Fanuc KAREL source: kc00004.KL

-- PROVISIONAL review KL for V1013-1; original PC SHA256 3c03b46ae540357a8fdae369b7eedd962a0a2d7ad2d21525eb34883495ea0831
-- Incomplete behavior may be omitted. Consult companion uncertainty JSON. Do not deploy.
PROGRAM KC00004
%NOLOCKGROUP
BEGIN
  -- UNRESOLVED_PC offsets 5-35; opcodes 27,22,22,22,2A,22,31
  -- UNRESOLVED_PC offsets 40-44; opcodes 7F
END KC00004
